/// machine data that is used through most sequences of the unit (motor speed, axes positions, ...)
TYPE MoverDataMachine :
STRUCT
  Slowspeed : LREAL;
  Highspeed : LREAL;
END_STRUCT
END_TYPE

(* stored: Version 1.1.0.1
   DUT MoverDataMachine: Id {fae4c575-0c3c-43f8-9959-77952c364550} *)
